(*
SPDX-FileCopyrightText: © 2026 Oleksandr Tiutyk <trofimich@gmail.com>
SPDX-License-Identifier: MIT
License: https://opensource.org/license/mit
*)

(*!
<summary>Exposes the captured native exception code alongside the common exception diagnostics.</summary>
<description>
The code identifies the captured native error, not the framework transport code used for propagation.
Obtaining this interface does not transfer ownership or extend the exception's lifetime.
</description>
*)

INTERFACE ISystemException EXTENDS IException

(*!
<summary>Returns the captured native exception code.</summary>
*)

{attribute 'monitoring' := 'call'}
PROPERTY ExceptionCode : __SYSTEM.ExceptionCode
GET
END_GET
END_PROPERTY

END_INTERFACE

(* stored: Version 1.1.0.1
   Itf ISystemException: Id {7870ea65-b79e-4a5f-a0cf-37b06b88ed45}
   Property ExceptionCode: Id {15970fe0-8365-4901-b4a4-73314108321e}
   Get Get: Id {5aed6761-fded-45fb-a3b9-33b86ea1a435} *)
